// Mitsubishi GX Works2 project: n04   PLC: Q02/Q02H

PROGRAM MAIN
VAR
  자기_1 : 자기;
  자기_2 : 자기;
  자기_3 : 자기;
  자기_4 : 자기;
END_VAR
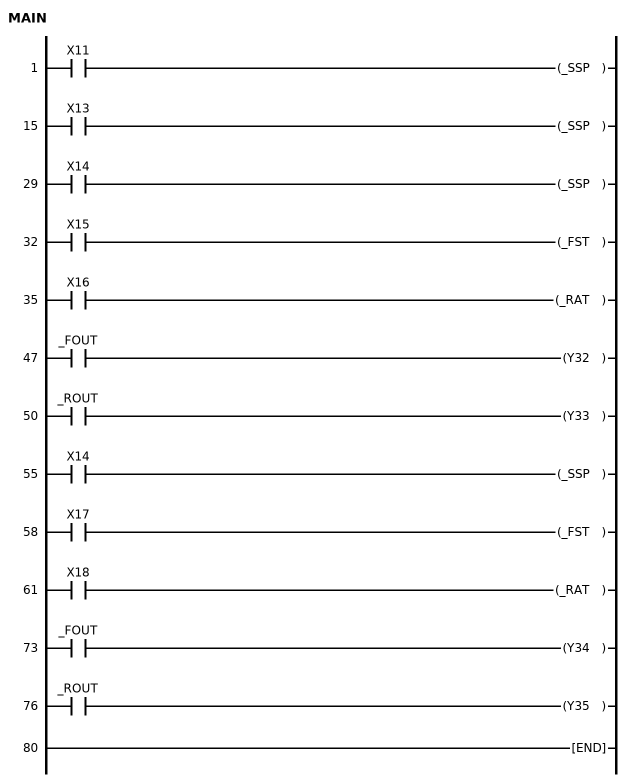
; FB BLK START 자기(자기_1)
1     LD      X11
      OUT     _SSP
; FB START
; FB_NAME 자기
; INSTANCE_NAME 자기_1
; FB IN_B:SSP
; FB OUT_FOUT:B
; FB IN_B:FST
; FB OUT_ROUT:B
; FB IN_B:RAT
; FB END
; FB BLK END
; FB BLK START 자기(자기_2)
15    LD      X13
      OUT     _SSP
; FB START
; FB_NAME 자기
; INSTANCE_NAME 자기_2
; FB IN_B:SSP
; FB OUT_FOUT:B
; FB IN_B:FST
; FB OUT_ROUT:B
; FB IN_B:RAT
; FB END
; FB BLK END
; FB BLK START 자기(자기_3)
29    LD      X14
      OUT     _SSP
32    LD      X15
      OUT     _FST
35    LD      X16
      OUT     _RAT
; FB START
; FB_NAME 자기
; INSTANCE_NAME 자기_3
; FB IN_B:SSP
; FB OUT_FOUT:B
; FB IN_B:FST
; FB OUT_ROUT:B
; FB IN_B:RAT
; FB END
47    LD      _FOUT
      OUT     Y32
50    LD      _ROUT
      OUT     Y33
; FB BLK END
; FB BLK START 자기(자기_4)
55    LD      X14
      OUT     _SSP
58    LD      X17
      OUT     _FST
61    LD      X18
      OUT     _RAT
; FB START
; FB_NAME 자기
; INSTANCE_NAME 자기_4
; FB IN_B:SSP
; FB OUT_FOUT:B
; FB IN_B:FST
; FB OUT_ROUT:B
; FB IN_B:RAT
; FB END
73    LD      _FOUT
      OUT     Y34
76    LD      _ROUT
      OUT     Y35
; FB BLK END
80    END
END_PROGRAM

FUNCTION_BLOCK 자기
VAR_INPUT
  SSP : BOOL;
  FST : BOOL;
END_VAR
VAR_OUTPUT
  FOUT : BOOL;
END_VAR
VAR_INPUT
  RAT : BOOL;
END_VAR
VAR_OUTPUT
  ROUT : BOOL;
END_VAR
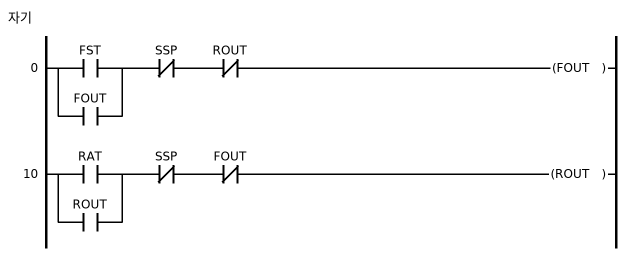
0     LD      FST
      OR      FOUT
      ANI     SSP
      ANI     ROUT
      OUT     FOUT
10    LD      RAT
      OR      ROUT
      ANI     SSP
      ANI     FOUT
      OUT     ROUT
END_FUNCTION_BLOCK
